TYPE TYP_VAC_GEN_HW :
STRUCT
	In : TYP_VAC_GEN_HW_IN;
	Out : TYP_VAC_GEN_HW_OUT;
END_STRUCT
END_TYPE

(* stored: Version 1.1.0.1, ProductVersion 3.1.4024.12
   DUT TYP_VAC_GEN_HW: Id {2c27e046-70fc-47d0-b57b-2675ee3c51dc} *)
